{attribute 'qualified_only'}
{attribute 'to_string'}
TYPE E_HandOverState:
(**************************************************************************************
 * 	Application		:	BoxControl Framework
 *	Revision		:	$Revision: 404529 $
 *	Revision date	:	$Date: 2018-04-23 08:21:38 +0200 (Mo., 23 Apr 2018) $
 *	Last changed by	:	$Author: b7bolm $
 *	URL				:	$URL: http://almscdc.swisslog.com/repo/SWPD/Development/BoxControlFramework/20_Release/trunk/01_Software/BCF/BCF/JumpStart/20_Product/10_App/12_E_Functions/10_Lib/10_Conv/10_Functions/01_DUTs/E_HandOverState.TcDUT $
 *
 *	Purpose			:	Handover states
 *
 * ------------------------------------------------------------------------------------
 *	Copyright Swisslog [IP AG], Switzerland. All rights reserved.
 * 
 * ------------------------------------------------------------------------------------
 *	
 * 	Revision History: 
 *
 * 	VERSION			DATE			INITIALS			DESCRIPTION
 *	0.1				01.01.2001		swl 				Example
 *
 **************************************************************************************)
(
	UNDEFINED			:= 0,
	IDLE				:= 1,
	READY				:= 2,
	ACTIVE				:= 3,
	STOP				:= 4,
	INTERRUPTED			:= 5,
	COMPLETE			:= 6
);
END_TYPE

(* stored: Version 1.1.0.1, ProductVersion 3.1.4024.4
   DUT E_HandOverState: Id {49f7259f-f264-4de8-b395-3eccda1e924e} *)
